{attribute 'linkalways'} 
{attribute 'no_explicit_call' := 'This FB is a CLASS and must be accessed using methods or properties'}
{attribute 'enable_dynamic_creation'}
FUNCTION_BLOCK Node_F_VN_DrawLine_TcVnVector4_LREAL EXTENDS VisionNode
VAR
    aLine : _TcVnVector4_LREAL;
    ipDestImage : _ITcVnImage;
    aColor : _TcVnVector4_LREAL;
    nThickness : _DINT(1);
    hrPrev : _HRESULT(S_OK);
	hresult : _HRESULT(S_OK);
END_VAR

METHOD PUBLIC  Clone : I_Node
VAR
	pNode : POINTER TO Node_F_VN_DrawLine_TcVnVector4_LREAL;
END_VAR
pNode := __NEW(Node_F_VN_DrawLine_TcVnVector4_LREAL);
Clone := pNode^;
END_METHOD

METHOD FB_init : BOOL
VAR_INPUT
	bInitRetains : BOOL; // if TRUE, the retain variables are initialized (warm start / cold start)
	bInCopyCode : BOOL;  // if TRUE, the instance afterwards gets moved into the copy code (online change)
END_VAR
AddInput('aLine', aLine);
AddInput('ipDestImage', ipDestImage);
AddInput('aColor', aColor);
AddInput('hrPrev', hrPrev);
AddOutput('ipDestImage', ipDestImage);
AddOutput('hresult',hresult);
AddParameter('nThickness', nThickness);
END_METHOD

METHOD PROTECTED OnExecute
hresult.Value := F_VN_DrawLine_TcVnVector4_LREAL(
    aLine := aLine.Value,
	ipDestImage := ipDestImage.Value,
    aColor := aColor.Value,
    nThickness := nThickness.Value,
	hrPrev:= hrPrev.Value);
END_METHOD

METHOD PUBLIC PreExecutionCheck
VAR_INPUT
	Check : I_PreExecutionChecks;
END_VAR
Check.IsTrue(ipDestImage.IsValid, 'ipDestImage must contain an image');
Check.IsTrue(nThickness.Value >= 1, 'nThickness must be greater than or equal to 1');
END_METHOD

END_FUNCTION_BLOCK

(* stored: Version 1.1.0.1, ProductVersion 3.1.4024.15
   POU Node_F_VN_DrawLine_TcVnVector4_LREAL: Id {110d1d30-d0e3-07d2-17fb-66b7772746b7}, SpecialFunc None
   Folder Constructor: Id {827bea5f-61ba-040b-2195-07851c8d53ee}
   Method Clone: Id {18e5f27a-e1ed-02e2-3062-0cc95da0e5b7}
   Method FB_init: Id {d0af5d35-428e-05b6-336f-19b98dde0307}
   Method OnExecute: Id {a3cdf037-404e-02af-16df-fab0e9f8a499}
   Method PreExecutionCheck: Id {3147cdf1-2028-0afa-354f-9467005e203b} *)
